(* PLC project Unnamed, Unknown Unnamed 1 *)
(* stored: creationDateTime 2026-02-02T14:07:16, modificationDateTime 2026-02-02T14:07:16 *)

FUNCTION_BLOCK Circular_queue
  VAR_INPUT
    XPush : BOOL;
    XPop : BOOL;
    iInputVal : INT;
  END_VAR
  VAR_OUTPUT
    iOutputVal : INT;
    iCount : INT;
    Operation_Cost : INT;
  END_VAR
  VAR
    Buffer : ARRAY [0..4999] OF INT;
    Head : INT;
    Tail : INT;
    MaxLen : INT;
    R_Trig_Push : R_TRIG;
    R_Trig_Pop : R_TRIG;
  END_VAR

            (* Edge Detection *)
R_Trig_Push(CLK := xPush);
R_Trig_Pop(CLK := xPop);

(* initialize MaxLen if 0 (safety check) *)
MaxLen := 5000;

(* --- PUSH (Enqueue) --- *)
IF R_Trig_Push.Q THEN
    (* Only push if not full (Optional safety, but good practice) *)
    IF iCount < MaxLen THEN
        Buffer[Head] := iInputVal;
        Head := Head + 1;
        IF Head >= MaxLen THEN Head := 0; END_IF;
        
        (* DIRECT COUNTING - The Fix *)
        iCount := iCount + 1; 
    END_IF;
END_IF;

(* --- POP (Dequeue) --- *)
IF R_Trig_Pop.Q AND iCount > 0 THEN
    iOutputVal := Buffer[Tail];
    Tail := Tail + 1;
    IF Tail >= MaxLen THEN Tail := 0; END_IF;
    
    (* DIRECT COUNTING - The Fix *)
    iCount := iCount - 1;
    Operation_Cost := 0; 
END_IF;
          
END_FUNCTION_BLOCK

FUNCTION_BLOCK FB_FIFO
  VAR_INPUT
    XPush : BOOL;
    XPop : BOOL;
    iInputVal : INT;
  END_VAR
  VAR_OUTPUT
    iOutputVal : INT;
    iCount : INT;
    Operation_Cost : INT;
  END_VAR
  VAR
    Buffer : ARRAY [0..4999] OF INT;
    i : INT;
    R_Trig_Push : R_TRIG;
    R_Trig_Pop : R_TRIG;
  END_VAR

            (* Edge Detection *)
R_Trig_Push(CLK := xPush);
R_Trig_Pop(CLK := xPop);

(* --- PUSH (FFL) --- *)
(* Simply add to the end. This part is actually fast (O(1)) *)
IF R_Trig_Push.Q AND iCount < 5000 THEN
    Buffer[iCount] := iInputVal;
    iCount := iCount + 1;
END_IF;

(* --- POP (FFU) - THE EXPENSIVE PART --- *)
(* This simulates the AB FFU shifting mechanism *)
IF R_Trig_Pop.Q AND iCount > 0 THEN
    
    (* 1. Grab the value at Head (Index 0) *)
    iOutputVal := Buffer[0];
    
    (* 2. THE SHIFT LOOP (The "Bad" Part) *)
    (* We must physically move every item down one slot *)
    (* If you have 50 items, this loop runs 49 times! *)
    
    FOR i := 0 TO iCount - 2 DO
        Buffer[i] := Buffer[i+1]; (* Move data from i+1 to i *)
        
        (* Increment the "Cost" Counter to visualize the inefficiency *)
        Operation_Cost := Operation_Cost + 1; 
    END_FOR;

    (* 3. Clear the last slot (optional, but clean) *)
    Buffer[iCount - 1] := 0;

    (* 4. Decrement Count *)
    iCount := iCount - 1;
    
END_IF;
          
END_FUNCTION_BLOCK

PROGRAM main
  VAR
    Output_Bad AT %QW1 : INT;
    Output_Good AT %QW4 : INT;
    Test_value AT %QW5 : INT;
    Queue_Count AT %QW0 : INT;
    Shift_Counter AT %QW3 : INT;
    Shift_Counter_Good AT %QW2 : INT;
  END_VAR
  VAR
    My_Bad_FIFO : FB_FIFO;
    My_Good_FIFO : CIRCULAR_QUEUE;
    pb_Push : BOOL;
    pb_Pop : BOOL;
    Input_Data : INT;
    Auto_TImer : TON;
    Test_Step : INT := 0;
    Auto_Start : BOOL := FALSE;
    Fill_Queue_Now : BOOL := FALSE;
    i : INT := 0;
    Queue_Count_Good : INT := 0;
  END_VAR

            (* ============================================================= *)
(* ZONE 1: THE STRESS TEST LOADER (Instant Fill) *)
(* ============================================================= *)
(* This logic only runs ONCE when you force 'Fill_Queue_Now' to TRUE. *)
(* It pauses the scan cycle, stuffs 5,000 items into the queues, *)
(* and then releases the PLC back to normal operation. *)

IF Fill_Queue_Now THEN
    
    (* Loop from 1 to 5000 to fill the array completely *)
    FOR i := 1 TO 5000 DO
        
        (* 1. SIMULATE RISING EDGE (Push Button Press) *)
        (* We call the FBs directly here to force the data in *)
        My_Bad_FIFO(xPush := TRUE, xPop := FALSE, iInputVal := i);
        My_Good_FIFO(xPush := TRUE, xPop := FALSE, iInputVal := i);
        
        (* 2. SIMULATE FALLING EDGE (Push Button Release) *)
        (* We must call them again with FALSE to reset the trigger for the next loop iteration *)
        My_Bad_FIFO(xPush := FALSE, xPop := FALSE, iInputVal := i);
        My_Good_FIFO(xPush := FALSE, xPop := FALSE, iInputVal := i);
        
    END_FOR;
    
    (* Reset the trigger so it doesn't run forever *)
    Fill_Queue_Now := FALSE;
    
END_IF;


(* ============================================================= *)
(* ZONE 2: NORMAL OPERATION (Manual Pop) *)
(* ============================================================= *)
(* This runs every single scan cycle. It listens to your manual *)
(* 'pb_Pop' button so you can trigger the unloads when ready. *)

(* Call the Bad FIFO (Linear Shift) *)
My_Bad_FIFO(
    xPush := pb_Push,      (* Normal button control *)
    xPop := pb_Pop,        (* Normal button control *)
    iInputVal := Input_Data,
    iOutputVal => Output_Bad,
    iCount => Queue_Count,
    Operation_Cost => Shift_Counter
);

(* Call the Good FIFO (Circular Buffer) *)
My_Good_FIFO(
    xPush := pb_Push,
    xPop := pb_Pop,
    iInputVal := Input_Data,
    iOutputVal => Output_Good,
    iCount => Queue_Count_Good,
    Operation_Cost => Shift_Counter_Good
);
          
END_PROGRAM

CONFIGURATION Config0
  RESOURCE Res0 ON PLC
    TASK task0(INTERVAL := T#20ms, PRIORITY := 1);
    PROGRAM instance0 WITH task0 : main;
  END_RESOURCE
END_CONFIGURATION
